// Axis Share data for sync operation with other blocks
INTERFACE I_MotionAxisShareData

PROPERTY ExecHome : BOOL
GET
END_GET
END_PROPERTY

PROPERTY ExecMove : BOOL
GET
END_GET
END_PROPERTY

PROPERTY HomeBusy : BOOL
SET
END_SET
END_PROPERTY

PROPERTY LimBackward : BOOL
GET
END_GET
END_PROPERTY

PROPERTY LimForward : BOOL
GET
END_GET
END_PROPERTY

PROPERTY LimHome : BOOL
GET
END_GET
END_PROPERTY

PROPERTY MoveBusy : BOOL
SET
END_SET
END_PROPERTY

PROPERTY NegativeDirection : BOOL
SET
END_SET
END_PROPERTY

PROPERTY PositiveDirection : BOOL
SET
END_SET
END_PROPERTY

PROPERTY ResetDone : BOOL
SET
END_SET
END_PROPERTY

PROPERTY RestoreDone : BOOL
SET
END_SET
END_PROPERTY

PROPERTY SavedPosition : LREAL
SET
END_SET
END_PROPERTY

END_INTERFACE

(* stored: Version 1.1.0.1
   Itf I_MotionAxisShareData: Id {3731b878-8d4c-43b9-8fcd-40a9246a4c02}
   Property ExecHome: Id {7c3f7ac5-8ea0-46fc-9fd8-badb79fd280f}
   Get Get: Id {bb3f4c48-927f-4bd7-9ce2-b367a7c28297}
   Property ExecMove: Id {3538d87e-62f5-4e43-8409-49f36e6f0022}
   Get Get: Id {e46c7197-07ab-4c11-b123-454734665f3f}
   Property HomeBusy: Id {da9f3c2b-5921-442c-ba90-324a2d22b131}
   Set Set: Id {7a7f2453-52bf-446e-be4e-bf32ac291d8c}
   Property LimBackward: Id {26de73e5-5da0-4b40-bb73-0419302b2a81}
   Get Get: Id {31214624-1888-45ee-981d-984b06dbdd8f}
   Property LimForward: Id {7ce553ec-4c68-4824-b41d-aedea8a39929}
   Get Get: Id {2c2043cc-598a-48dd-8d7a-404d6ff7f552}
   Property LimHome: Id {5703ca74-1136-4580-87fc-34cb390d97f1}
   Get Get: Id {ec705d9c-959b-4fc7-8de7-976e1c397092}
   Property MoveBusy: Id {cb822bd0-33f7-4bb0-94ff-bb6844da17c8}
   Set Set: Id {42cadb91-27db-401b-8b52-0815c59fdd03}
   Property NegativeDirection: Id {e29497a5-1673-4757-bf97-dc4101219cf8}
   Set Set: Id {1ddceb5c-7126-4132-8dab-771bdb4e8509}
   Property PositiveDirection: Id {5773dff0-b318-4b19-a704-d1c48659ab24}
   Set Set: Id {17d6efe1-f492-4dfb-a1c2-b6870b2fe1f9}
   Property ResetDone: Id {b6933acc-1da2-4f64-9cc3-54287f2e8bba}
   Set Set: Id {a0f59ab1-81b1-41fb-bcc5-122f855cfe3d}
   Property RestoreDone: Id {79bfcbbe-cafa-4936-95fb-4b97cfcfbb24}
   Set Set: Id {486a82a1-77a6-4fc4-8ec2-1b1b2d5a8f5f}
   Property SavedPosition: Id {d50c808e-413b-4e8c-a493-6812442d0fdf}
   Set Set: Id {0a9fc5b8-7c83-472c-ba94-febe0c2a1ed1} *)
